FUNCTION_BLOCK FlushSelector (* CAT Function Block Type *)
  (* Standard: 61499-2 *)
  (* Version 0.0, 6/22/2026, Schneider Electric, template *)
  PACKAGE SE.Nereda;
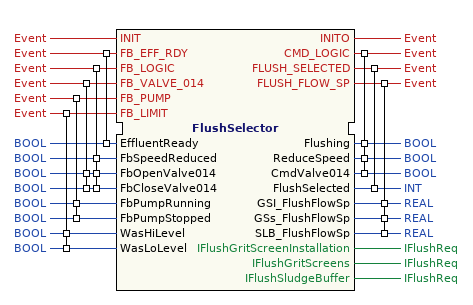
  EVENT_INPUT
    INIT;
    FB_EFF_RDY WITH EffluentReady;
    FB_LOGIC WITH FbSpeedReduced, FbOpenValve014, FbCloseValve014;
    FB_VALVE_014 WITH FbOpenValve014, FbCloseValve014;
    FB_PUMP WITH FbPumpRunning, FbPumpStopped;
    FB_LIMIT WITH WasHiLevel, WasLoLevel;
  END_EVENT
  EVENT_OUTPUT
    INITO;
    CMD_LOGIC WITH ReduceSpeed, CmdValve014, Flushing;
    FLUSH_SELECTED WITH FlushSelected; (* Execution Confirmation *)
    FLUSH_FLOW_SP WITH GSI_FlushFlowSp, GSs_FlushFlowSp, SLB_FlushFlowSp;
  END_EVENT
  VAR_INPUT
    EffluentReady : BOOL;
    FbSpeedReduced : BOOL;
    FbOpenValve014 : BOOL;
    FbCloseValve014 : BOOL;
    FbPumpRunning : BOOL;
    FbPumpStopped : BOOL;
    WasHiLevel : BOOL;
    WasLoLevel : BOOL;
  END_VAR
  VAR_OUTPUT
    Flushing : BOOL;
    ReduceSpeed : BOOL;
    CmdValve014 : BOOL;
    FlushSelected : INT;
    GSI_FlushFlowSp : REAL;
    GSs_FlushFlowSp : REAL;
    SLB_FlushFlowSp : REAL;
  END_VAR
  PLUGS
    IFlushGritScreenInstallation : IFlushReq;
    IFlushGritScreens : IFlushReq;
    IFlushSludgeBuffer : IFlushReq;
  END_PLUGS
  (* 01 - FUNCTIONNAL INPUT INTERFACE *)
  (* 00 - INITIALIZATION *)
  (* 05 - LOGIC *)
  (* 06 - HMI INTERFACE *)
  (* 03 - FIELD INTERFACE *)
  (* Flush Selector *)
  (* 02 - FUNCTIONNAL OUTPUT INTERFACE *)
  (* Cycle *)
  FBS
    FlushSelector : FlushingSelector;
    IThis : FlushSelector_HMI(QI := TRUE);
    ReqFlush_Cycle : E_CYCLE(DT := T#1s);
    FlushEvent : E_MERGE;
    EO_FLUSH_FLOW_SP : E_MERGE_4;
    EffluentReday : AND_88A3DD8EC65DD11C; {SET_ATTRIBUTE(Configuration.GenericFBType.InterfaceParams, Runtime.Standard#CNT:=2;OUT:BOOL)}
    FB1 : E_MERGE;
    FB2 : IntValueChanged;
    Wait : E_DELAY(DT := T#1s);
  END_FBS
  EVENT_CONNECTIONS
    ReqFlush_Cycle.EO TO FlushEvent.EI1;
    FlushSelector.C5198EBE6703874F TO ReqFlush_Cycle.START;
    FlushSelector.B482DC569AD88DF9 TO ReqFlush_Cycle.STOP;
    FB_VALVE_014 TO IFlushGritScreenInstallation.158ACCEF11EA11F4;
    FB_PUMP TO IFlushGritScreenInstallation.158ACCEF11EA11F4;
    FB_VALVE_014 TO IFlushGritScreens.158ACCEF11EA11F4;
    FB_PUMP TO IFlushGritScreens.158ACCEF11EA11F4;
    FB_VALVE_014 TO IFlushSludgeBuffer.158ACCEF11EA11F4;
    FB_PUMP TO IFlushSludgeBuffer.158ACCEF11EA11F4;
    FlushSelector.C5198EBE6703874F TO FB1.EI1;
    EO_FLUSH_FLOW_SP.EO TO FLUSH_FLOW_SP;
    IFlushGritScreenInstallation.A591EFC748C65FB0 TO EO_FLUSH_FLOW_SP.EI1;
    IFlushGritScreens.A591EFC748C65FB0 TO EO_FLUSH_FLOW_SP.EI2;
    IFlushSludgeBuffer.A591EFC748C65FB0 TO EO_FLUSH_FLOW_SP.EI3;
    FlushSelector.B482DC569AD88DF9 TO FlushEvent.EI2;
    FB_EFF_RDY TO EffluentReday.REQ;
    FlushEvent.EO TO FlushSelector.D8D7EDABEA7B3922;
    INIT TO IThis.914030477D815D8C;
    IFlushGritScreenInstallation.91C62E5F9EC3AD97 TO IThis.B10EF0CE55004EDB;
    IFlushGritScreens.91C62E5F9EC3AD97 TO IThis.B10EF0CE55004EDB;
    IFlushSludgeBuffer.91C62E5F9EC3AD97 TO IThis.B10EF0CE55004EDB;
    IThis.A86ED5016CE18720 TO INITO;
    IFlushGritScreenInstallation.91C62E5F9EC3AD97 TO FlushSelector.B3C3778B51CB7C0B;
    IFlushGritScreens.91C62E5F9EC3AD97 TO FlushSelector.B3C3778B51CB7C0B;
    IFlushSludgeBuffer.91C62E5F9EC3AD97 TO FlushSelector.B3C3778B51CB7C0B;
    IFlushGritScreenInstallation.058C8BB5EF4C4954 TO FlushEvent.EI2;
    IFlushGritScreens.058C8BB5EF4C4954 TO FlushEvent.EI2;
    IFlushSludgeBuffer.058C8BB5EF4C4954 TO FlushEvent.EI2;
    EffluentReday.CNF TO CMD_LOGIC;
    FlushSelector.72F6AA492327E76C TO EffluentReday.REQ;
    FB_LOGIC TO IFlushGritScreenInstallation.158ACCEF11EA11F4;
    FB_LOGIC TO IFlushGritScreens.158ACCEF11EA11F4;
    FB_LOGIC TO IFlushSludgeBuffer.158ACCEF11EA11F4;
    FB_LIMIT TO IFlushGritScreenInstallation.158ACCEF11EA11F4;
    FB_LIMIT TO IFlushGritScreens.158ACCEF11EA11F4;
    FB_LIMIT TO IFlushSludgeBuffer.158ACCEF11EA11F4;
    FB1.EO TO FLUSH_SELECTED;
    FlushSelector.72F6AA492327E76C TO FB2.77F8F9CFF707DAFF;
    FB2.93AE3729A9342678 TO FB1.EI2;
    FlushSelector.02F68A5DD7B717EF TO Wait.START;
    Wait.EO TO FlushSelector.DE111E414B61F07B;
  END_CONNECTIONS
  DATA_CONNECTIONS
    IFlushGritScreenInstallation.B5CD30493D22784A TO FlushSelector.DB000855E101C77F;
    IFlushGritScreenInstallation.78ED129B4768A8A1 TO FlushSelector.0E98C03A6F673D7F;
    IFlushGritScreenInstallation.23612E77D592C190 TO FlushSelector.9DEF7B7D7715E0CE;
    IFlushGritScreens.78ED129B4768A8A1 TO FlushSelector.91C603F64C0C70F5;
    IFlushGritScreens.23612E77D592C190 TO FlushSelector.CCDB4DBCA0B4B23D;
    IFlushSludgeBuffer.78ED129B4768A8A1 TO FlushSelector.998C0B5D38D41A44;
    IFlushSludgeBuffer.23612E77D592C190 TO FlushSelector.4AFA863861C84038;
    EffluentReady TO EffluentReday.IN1;
    EffluentReday.OUT TO Flushing;
    FlushSelector.E35DB6B1DD2B2E36 TO ReduceSpeed;
    FlushSelector.D74C26B56D3ECE0D TO CmdValve014;
    FbOpenValve014 TO IFlushGritScreenInstallation.309BBEDA7DF51DE0;
    FbCloseValve014 TO IFlushGritScreenInstallation.E3447F193E0C5923;
    FbPumpRunning TO IFlushGritScreenInstallation.102FEFFE81A835E5;
    FbPumpStopped TO IFlushGritScreenInstallation.32E78DF7D9CBD985;
    FbOpenValve014 TO IFlushGritScreens.309BBEDA7DF51DE0;
    FbCloseValve014 TO IFlushGritScreens.E3447F193E0C5923;
    FbPumpRunning TO IFlushGritScreens.102FEFFE81A835E5;
    FbPumpStopped TO IFlushGritScreens.32E78DF7D9CBD985;
    FbOpenValve014 TO IFlushSludgeBuffer.309BBEDA7DF51DE0;
    FbCloseValve014 TO IFlushSludgeBuffer.E3447F193E0C5923;
    FbPumpRunning TO IFlushSludgeBuffer.102FEFFE81A835E5;
    FbPumpStopped TO IFlushSludgeBuffer.32E78DF7D9CBD985;
    FB2.AA81B8787A42C5C8 TO FlushSelected;
    IFlushGritScreenInstallation.34B76CCA964D89EE TO GSI_FlushFlowSp;
    IFlushGritScreens.34B76CCA964D89EE TO GSs_FlushFlowSp;
    IFlushSludgeBuffer.34B76CCA964D89EE TO SLB_FlushFlowSp;
    IFlushGritScreenInstallation.B5CD30493D22784A TO IThis.910D6147A55B7609;
    FB2.AA81B8787A42C5C8 TO IThis.64971CE4161C8DDB;
    IFlushGritScreens.B5CD30493D22784A TO FlushSelector.6F16CF1994B563D7;
    IFlushSludgeBuffer.B5CD30493D22784A TO FlushSelector.DB568F49C4639AC9;
    FlushSelector.90BE0054E7DD7D45 TO EffluentReday.IN2;
    IFlushGritScreenInstallation.10050E1891596878 TO FlushSelector.D29FDD994529B71F;
    IFlushGritScreens.10050E1891596878 TO FlushSelector.2527676400CBF5ED;
    IFlushSludgeBuffer.10050E1891596878 TO FlushSelector.103BE80FBAF0C7F9;
    FbSpeedReduced TO IFlushGritScreenInstallation.0154EF4D281C90FC;
    FbSpeedReduced TO IFlushGritScreens.0154EF4D281C90FC;
    FbSpeedReduced TO IFlushSludgeBuffer.0154EF4D281C90FC;
    IFlushGritScreens.B5CD30493D22784A TO IThis.5B95BCAAAEA86F1D;
    IFlushSludgeBuffer.B5CD30493D22784A TO IThis.91935B7F69196492;
    WasHiLevel TO IFlushGritScreenInstallation.F75B2D6279DB7772;
    WasHiLevel TO IFlushGritScreens.F75B2D6279DB7772;
    WasHiLevel TO IFlushSludgeBuffer.F75B2D6279DB7772;
    WasLoLevel TO IFlushGritScreenInstallation.FBD19C5680BE3A13;
    WasLoLevel TO IFlushGritScreens.FBD19C5680BE3A13;
    WasLoLevel TO IFlushSludgeBuffer.FBD19C5680BE3A13;
    FlushSelector.CCD69D3E6C0C119E TO FB2.25B5287A5784F3EC;
  END_CONNECTIONS
END_FUNCTION_BLOCK
